// SIMATIC S7-200 project (STEP 7-Micro/WIN), CPU 222 REL 02.01

SYMBOL_TABLE USR1
AcionCxG         I0.0
AcionCxP         I0.1
S1               I0.2
S2               I0.3
S3               I0.4
S4               I0.5
S5               I1.6
S6               I0.6
S7               I0.7
S8               I1.0
S9               I1.1
EST1             Q0.0
EST2             Q0.1
CxG              Q0.2
CxP              Q0.3
VA1              Q0.4
VA1C             I1.2
VA1E             I1.3
V1E              Q1.0
V1S              Q1.1
V2E              Q1.2
V2S              Q1.3
AGUA_1           AIW0
AGUA_2           AIW2
VOL1             VD70
VOL2             VD100
REF1             VD110
REF2             VD120
E0               M0.0
E1               M0.1
E2               M0.2
E3               M0.3
E4               M0.4
E5               M0.5
E6               M0.6
E7               M0.7
E8               M1.0
E9               M1.1
E10              M1.2
E11              M1.3
E12              M1.4
END_SYMBOL_TABLE

ORGANIZATION_BLOCK MAIN:OB1
TITLE=POU Comment
BEGIN
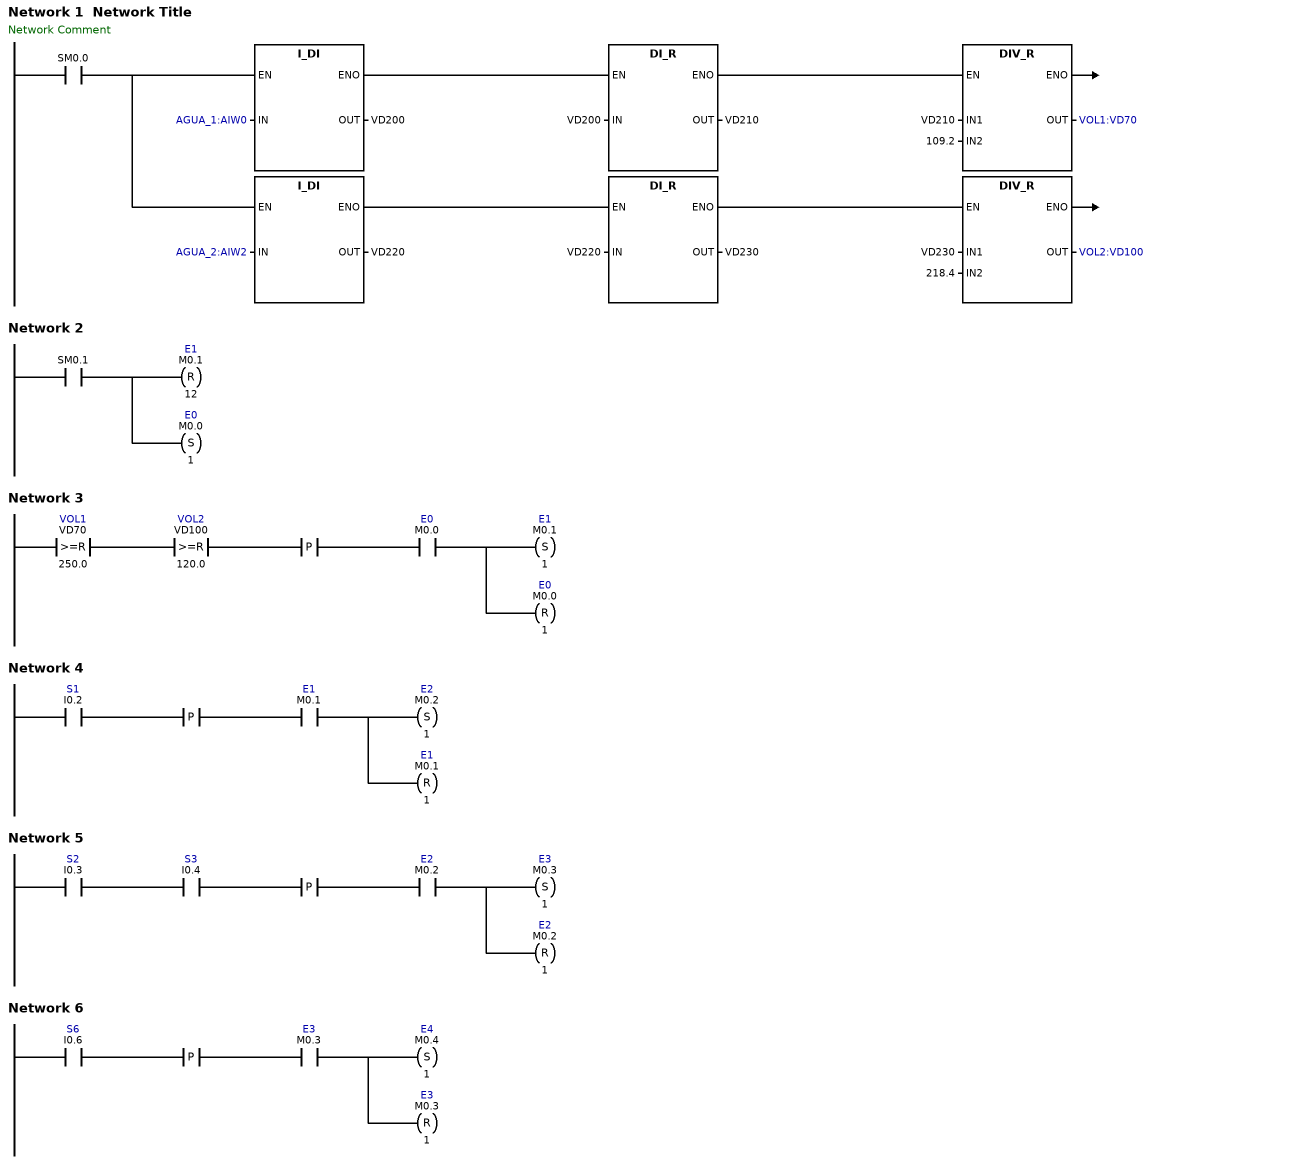
Network 1 // Network Title
// Network Comment
// (network saved uncompiled; LAD cells follow)
// row 0: c0 -| |- SM0.0 v  c1 --  c2 [I_DI EN:=power@row0, IN:=AGUA_1:AIW0, ENO=>power, OUT=>VD200]  c3 --  c4 --  c5 [DI_R EN:=power@row0, IN:=VD200, ENO=>power, OUT=>VD210]  c6 --  c7 --  c8 [DIV_R EN:=power@row0, IN1:=VD210, IN2:=109.2, ENO=>power, OUT=>VOL1:VD70]  c9 ->
// row 1: c0 ^v  c2 [box]  c5 [box]  c8 [box]
// row 2: c0 ^  c1 --  c2 [I_DI EN:=power@row2, IN:=AGUA_2:AIW2, ENO=>power, OUT=>VD220]  c3 --  c4 --  c5 [DI_R EN:=power@row2, IN:=VD220, ENO=>power, OUT=>VD230]  c6 --  c7 --  c8 [DIV_R EN:=power@row2, IN1:=VD230, IN2:=218.4, ENO=>power, OUT=>VOL2:VD100]  c9 ->
// row 3: c2 [box]  c5 [box]  c8 [box]
Network 2
LD     SM0.1
R      E1:M0.1, 12
S      E0:M0.0, 1
Network 3
LDR>=  VOL1:VD70, 250.0
AR>=   VOL2:VD100, 120.0
EU
A      E0:M0.0
S      E1:M0.1, 1
R      E0:M0.0, 1
Network 4
LD     S1:I0.2
EU
A      E1:M0.1
S      E2:M0.2, 1
R      E1:M0.1, 1
Network 5
LD     S2:I0.3
A      S3:I0.4
EU
A      E2:M0.2
S      E3:M0.3, 1
R      E2:M0.2, 1
Network 6
LD     S6:I0.6
EU
A      E3:M0.3
S      E4:M0.4, 1
R      E3:M0.3, 1
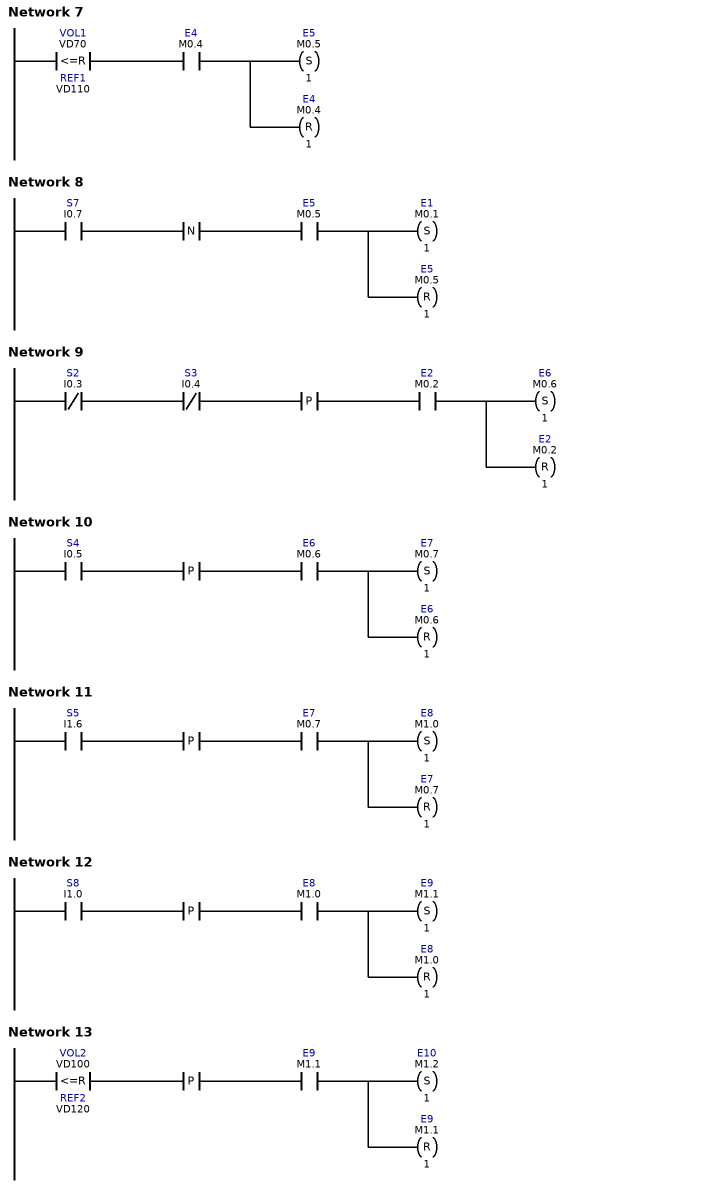
Network 7
LDR<=  VOL1:VD70, REF1:VD110
A      E4:M0.4
S      E5:M0.5, 1
R      E4:M0.4, 1
Network 8
LD     S7:I0.7
ED
A      E5:M0.5
S      E1:M0.1, 1
R      E5:M0.5, 1
Network 9
LDN    S2:I0.3
AN     S3:I0.4
EU
A      E2:M0.2
S      E6:M0.6, 1
R      E2:M0.2, 1
Network 10
LD     S4:I0.5
EU
A      E6:M0.6
S      E7:M0.7, 1
R      E6:M0.6, 1
Network 11
LD     S5:I1.6
EU
A      E7:M0.7
S      E8:M1.0, 1
R      E7:M0.7, 1
Network 12
LD     S8:I1.0
EU
A      E8:M1.0
S      E9:M1.1, 1
R      E8:M1.0, 1
Network 13
LDR<=  VOL2:VD100, REF2:VD120
EU
A      E9:M1.1
S      E10:M1.2, 1
R      E9:M1.1, 1
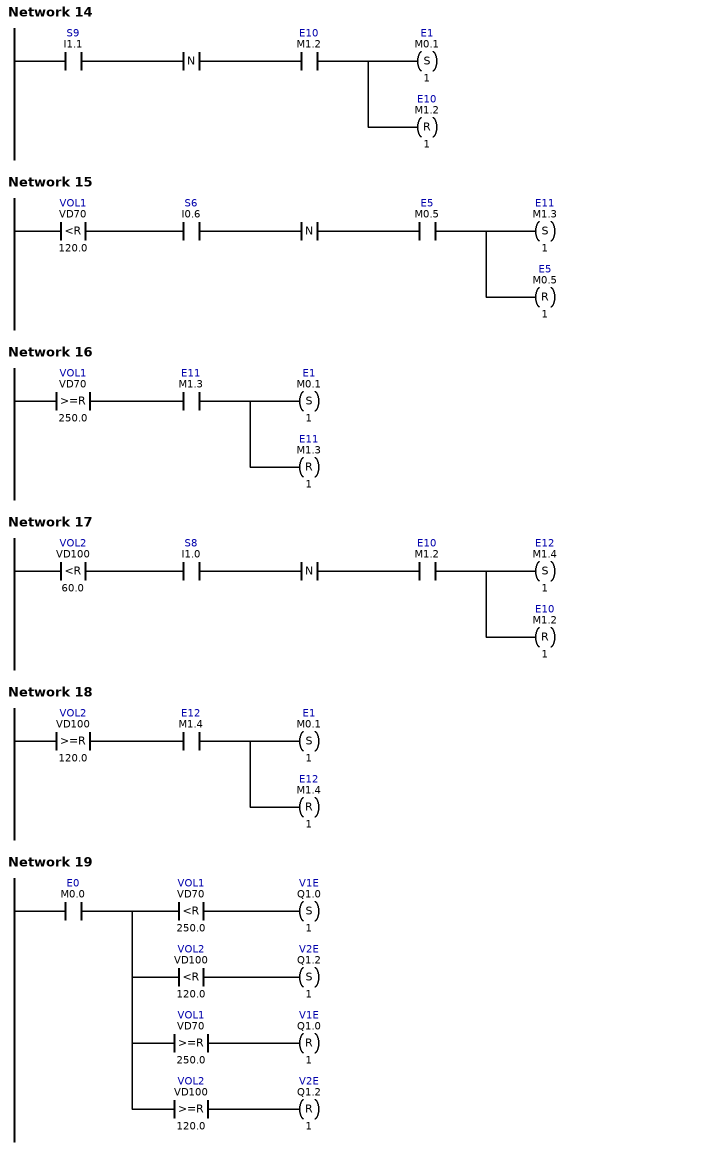
Network 14
LD     S9:I1.1
ED
A      E10:M1.2
S      E1:M0.1, 1
R      E10:M1.2, 1
Network 15
LDR<   VOL1:VD70, 120.0
A      S6:I0.6
ED
A      E5:M0.5
S      E11:M1.3, 1
R      E5:M0.5, 1
Network 16
LDR>=  VOL1:VD70, 250.0
A      E11:M1.3
S      E1:M0.1, 1
R      E11:M1.3, 1
Network 17
LDR<   VOL2:VD100, 60.0
A      S8:I1.0
ED
A      E10:M1.2
S      E12:M1.4, 1
R      E10:M1.2, 1
Network 18
LDR>=  VOL2:VD100, 120.0
A      E12:M1.4
S      E1:M0.1, 1
R      E12:M1.4, 1
Network 19
LD     E0:M0.0
LPS
AR<    VOL1:VD70, 250.0
S      V1E:Q1.0, 1
LRD
AR<    VOL2:VD100, 120.0
S      V2E:Q1.2, 1
LRD
AR>=   VOL1:VD70, 250.0
R      V1E:Q1.0, 1
LPP
AR>=   VOL2:VD100, 120.0
R      V2E:Q1.2, 1
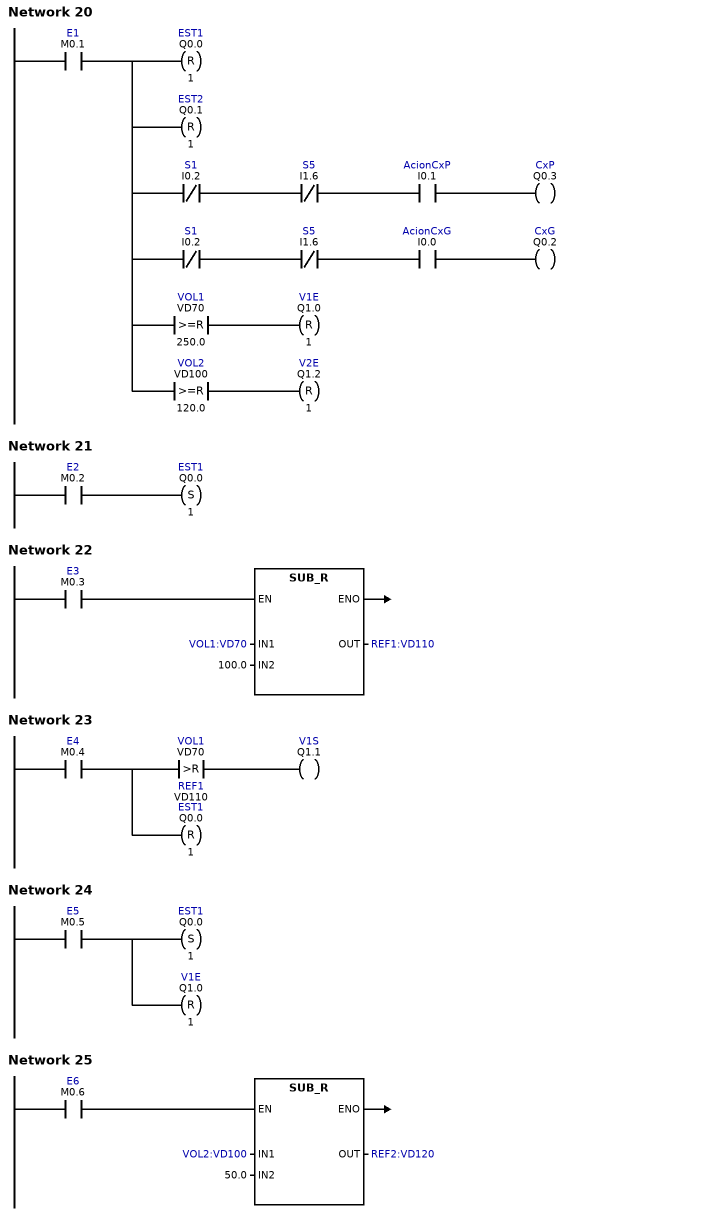
Network 20
LD     E1:M0.1
LPS
R      EST1:Q0.0, 1
R      EST2:Q0.1, 1
AN     S1:I0.2
AN     S5:I1.6
A      AcionCxP:I0.1
=      CxP:Q0.3
LRD
AN     S1:I0.2
AN     S5:I1.6
A      AcionCxG:I0.0
=      CxG:Q0.2
LRD
AR>=   VOL1:VD70, 250.0
R      V1E:Q1.0, 1
LPP
AR>=   VOL2:VD100, 120.0
R      V2E:Q1.2, 1
Network 21
LD     E2:M0.2
S      EST1:Q0.0, 1
Network 22
LD     E3:M0.3
MOVR   VOL1:VD70, REF1:VD110
-R     100.0, REF1:VD110
Network 23
LD     E4:M0.4
LPS
AR>    VOL1:VD70, REF1:VD110
=      V1S:Q1.1
LPP
R      EST1:Q0.0, 1
Network 24
LD     E5:M0.5
S      EST1:Q0.0, 1
R      V1E:Q1.0, 1
Network 25
LD     E6:M0.6
MOVR   VOL2:VD100, REF2:VD120
-R     50.0, REF2:VD120
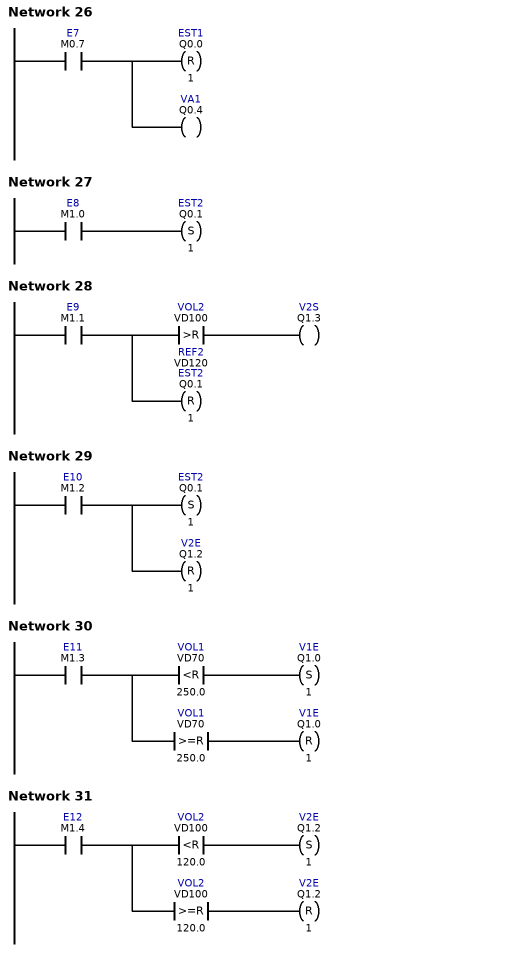
Network 26
LD     E7:M0.7
R      EST1:Q0.0, 1
=      VA1:Q0.4
Network 27
LD     E8:M1.0
S      EST2:Q0.1, 1
Network 28
LD     E9:M1.1
LPS
AR>    VOL2:VD100, REF2:VD120
=      V2S:Q1.3
LPP
R      EST2:Q0.1, 1
Network 29
LD     E10:M1.2
S      EST2:Q0.1, 1
R      V2E:Q1.2, 1
Network 30
LD     E11:M1.3
LPS
AR<    VOL1:VD70, 250.0
S      V1E:Q1.0, 1
LPP
AR>=   VOL1:VD70, 250.0
R      V1E:Q1.0, 1
Network 31
LD     E12:M1.4
LPS
AR<    VOL2:VD100, 120.0
S      V2E:Q1.2, 1
LPP
AR>=   VOL2:VD100, 120.0
R      V2E:Q1.2, 1
END_ORGANIZATION_BLOCK
